// Mitsubishi GX Developer project: C-2-1   PLC: FX2N

PROGRAM Main
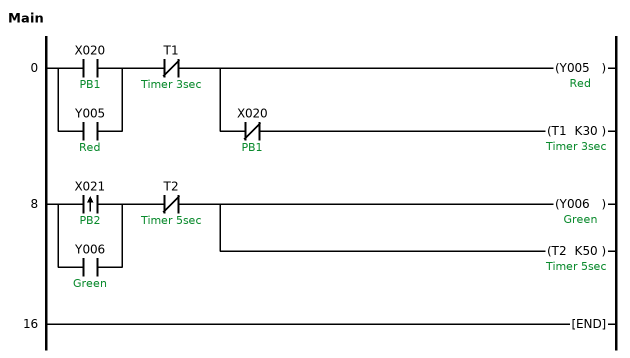
0     LD      X020  ; PB1
      OR      Y005  ; Red
      ANI     T1  ; Timer 3sec
      OUT     Y005  ; Red
      ANI     X020  ; PB1
      OUT     T1 K30  ; Timer 3sec
8     LDP     X021  ; PB2
      OR      Y006  ; Green
      ANI     T2  ; Timer 5sec
      OUT     Y006  ; Green
      OUT     T2 K50  ; Timer 5sec
16    END
END_PROGRAM
